FUNCTION_BLOCK NodeTriggerExtension EXTENDS ExtensionBase IMPLEMENTS I_EventHandler
VAR
	parent : I_Node;
	nodeInput_Trigger : InputPort_Trigger('trigger','HRESULT',THIS^);
	nodeOutput_Trigger : OutputPort('result','HRESULT',THIS^);
END_VAR

METHOD FB_exit : BOOL
VAR_INPUT
	bInCopyCode : BOOL; // if TRUE, the exit method is called for exiting an instance that is copied afterwards (online change).
END_VAR
IF bInCopyCode THEN
	RETURN;
END_IF

UnregisterWithParent();
END_METHOD

METHOD FB_init : BOOL
VAR_INPUT
	bInitRetains : BOOL; // if TRUE, the retain variables are initialized (warm start / cold start)
	bInCopyCode : BOOL;  // if TRUE, the instance afterwards gets moved into the copy code (online change)
	Name : T_MAXSTRING;
	Parent : I_Node;
END_VAR
THIS^.parent := Parent;
RegisterWithParent();
END_METHOD

METHOD PUBLIC HandleEvent
VAR_INPUT
	Event : I_Event;
END_VAR
{warning 'This needs to be implemented'}
END_METHOD

METHOD PROTECTED RegisterWithParent
VAR_INPUT
END_VAR
IF parent = 0 THEN
	RETURN;
END_IF

parent.AddExtension(THIS^);
END_METHOD

METHOD PROTECTED UnregisterWithParent
VAR_INPUT
END_VAR
IF parent = 0 THEN
	RETURN;
END_IF
END_METHOD

END_FUNCTION_BLOCK

(* stored: Version 1.1.0.1, ProductVersion 3.1.4024.12
   POU NodeTriggerExtension: Id {33e0a2d7-9483-08c7-064c-13c37845f3c6}, SpecialFunc None
   Folder Constructor: Id {ede2f570-9df8-03ad-3f5d-9c9a6b23db22}
   Folder Destructor: Id {f9bb0db8-25f5-04cb-3fad-e1dd95a9193b}
   Folder Protected: Id {eac92252-fb76-0f6f-076f-07b51cf3bcc3}
   Method FB_exit: Id {0976737d-d648-0a05-3fe5-2805e42e0e5a}
   Method FB_init: Id {552aaaf2-c686-0d38-32c4-997aac180a0c}
   Method HandleEvent: Id {425c6d59-f4b3-0dfd-36e8-c98c705cef2a}
   Method RegisterWithParent: Id {fe73466f-9102-0cc2-0083-a78a8d592deb}
   Method UnregisterWithParent: Id {875f0b67-3383-09e1-0c65-fe05d6b3969e} *)
